FUNCTION_BLOCK FB_Ramp
VAR_INPUT
	bEnableRamp : BOOL;
	fHeight : LREAL;
	fRampTime : LREAL;
	fInitialPos : LREAL;
	fMaxSpeed : LREAL;
END_VAR
VAR_OUTPUT
	fXRef : LREAL;
	fXDotRef : LREAL;
END_VAR
VAR
END_VAR


IF fRampTime > G_OPC.fMotionTime THEN
	fXDotRef := fHeight / fRampTime;
ELSE
	fXDotRef := 0.0;
END_IF

fXRef := fInitialPos + fHeight;

END_FUNCTION_BLOCK

(* stored: Version 1.1.0.1
   POU FB_Ramp: Id {0aea8e66-d7a8-409b-9f89-3625b52daf60}, SpecialFunc None *)
